PROGRAM MAIN
VAR		
	startdata 				AT %I* : UINT;	

	fbDemoAcyclic :			FB_SICK_WF_A70_EC;
	fbDemoProcesData :		FB_SICK_WF_A70_PB;
	structSick : 			ST_SICK_WF_A70;
	
	risingEdgeSignalRead : 		R_TRIG;
	risingEdgeSignalWrite :		R_TRIG;
	
	//Start read request
	xStartRead :			BOOL;
	
	//Start write request
	xStartWrite : 			BOOL;
	
	//Request done
	xDone :					BOOL;
	
END_VAR


risingEdgeSignalRead(CLK := xStartRead);
risingEdgeSignalWrite(CLK := xStartWrite);

TEEEEESSTTTTTTTTTTTTT


structSick.Selection.AutoDeSelect := TRUE;

IF risingEdgeSignalRead.Q AND NOT fbDemoAcyclic.Busy THEN
	xDone := FALSE;
	structSick.Selection.ProductID := TRUE;
	structSick.Selection.VendorName := TRUE;
	structSick.Selection.ProductName := TRUE;
	structSick.Selection.KeyLock := TRUE;
	structSick.Selection.SwitchpointBDC1Q1.All := TRUE;
	
	fbDemoAcyclic.RW := FALSE; //Read
	fbDemoAcyclic.Req := TRUE; //Start job
	
	(*Parameter write*)
ELSIF risingEdgeSignalWrite.Q AND NOT fbDemoAcyclic.Busy THEN
	// Init status
	xDone:= FALSE;

	// Parameter selection that should be written
	structSick.Selection.KeyLock:= TRUE;
	
	
	// Definition of the data that should be written 
	structSick.Data.KeyLock:= eKeylock;

	
	fbDemoAcyclic.RW:= TRUE; // Write
	fbDemoAcyclic.Req:= TRUE; // Start job
END_IF;
	

fbDemoAcyclic(
	NetID:= '10.25.60.57.3.3', 
	PortNumber:= 1, 
	TimeOut:= T#5S, 
	Done=> , 
	Busy=> , 
	Error=> , 
	ErrorCode=> , 
	MasterType:= eBECKHOFF_6224, 
	SlaveAddr:= 0, 
	Req:= , 
	RW:= TRUE, 
	DeviceData:= structSick);
	
	fbDemoAcyclic.Req := FALSE;
	
	IF fbDemoAcyclic.Done THEN
		xDone := TRUE;
	END_IF

END_PROGRAM

(* stored: Version 1.1.0.1, ProductVersion 3.1.4022.10
   POU MAIN: Id {59ebf7a5-a622-4e8e-b8cd-d8e3d4cc7dfa}, SpecialFunc None *)
